{attribute 'OPC.UA.DA.StructuredType' := '1'}
TYPE ST_SensorState :
STRUCT
	fValue 		: REAL; //status on / off
	sUnit		: STRING; //current unit of sensor value
END_STRUCT
END_TYPE

(* stored: Version 1.1.0.1, ProductVersion 3.1.4024.9
   DUT ST_SensorState: Id {2975f68f-a189-46c5-b8f3-10203fb5a404} *)
